// TIA Portal V15.1 export
// export: Created 2024-06-21T08:41:09.7541663Z, ExportSetting WithDefaults, DisplayName Totally Integrated Automation Portal, DisplayVersion V15.1 Update 5, DisplayName TIA Portal Openness, DisplayVersion V15.1 Update 5, DisplayName SINAMICS Startdrive Advanced, DisplayVersion V15.1, DisplayName G130, G150, S120, S150, SINAMICS MV, S210, DisplayVersion V15.1, DisplayName G110M, G120, G120C, G120D, G120P, DisplayVersion V15.1, DisplayName STEP 7 Professional, DisplayVersion V15.1 Update 5, DisplayName STEP 7 Safety, DisplayVersion V15.1, DisplayName WinCC Professional, DisplayVersion V15.1 Update 5, DisplayName SIMATIC Visualization Architect, DisplayVersion V15.1
FUNCTION "LGBLiftTable2Pos1S3Det-MoviFitFCPN-Config" : Void   // FC6651, FBD
TITLE = LMovUnit2Pos2Det2W2S-G120CU240PN-Config / LConfigMovUnit2Pos2W2S-G120PN / LGBLiftTable2Pos1S4Det-MoviFitFCPN-Config
{ S7_Optimized_Access := 'TRUE' }
AUTHOR : VCC
FAMILY : Control
NAME : Bit2Word
VERSION : 1.0
// =============================================================================
// Moves Configuration
// =============================================================================
// stored: AutoNumber false, IsIECCheckEnabled false, SetENOAutomatically False, UDAEnableTagReadback false
   VAR_INPUT
      C_ForceManual : Bool;   // Force Manual Enabled
      C_PosSetCheckUsed : Bool;   // 2nd Set Pos Check Used
      C_PosResCheckUsed : Bool;   // 2nd Set Pos Check Used
      C_AlarmResetUsed : Bool;   // Set position / If true, the Alarms will be stored untill reseted
      C_EnableMemBegin : Bool;   // Reset position / Enable memory Begin (Command Request is memorised until pos reached)
      C_EnIntlkAlm : Bool;   // Active / Enable interlock Alarm
      C_KeepPosition : Bool;   // Invisible / If true, the last position shall be kept ON and checked
      C_EnAlmDet : Bool;   // Object out of use / Enable Alarm
      C_EnableAlarmHW : Bool;   // Enable Alarm hardware (e.g. safetyswitch, motorprotector, detections)
      C_MotorProtectionNc : Bool;   // Motor Protection NC contact
      C_MotorProtectionUsed : Bool;   // Motor Protection used
      C_ReleaseBrakeUsed : Bool;   // Release brake used
      C_MotionStopUsed : Bool;   // Motion Stop used
      C_EnAlmOvertime : Bool;   // Interlock for Reset direction / Enable Overtime Alarm
      C_AlarmHighSeverity : Bool;   // Interlock alarm for Set direction / Alarm severity
      C_InitDirection : Bool;   // Initial direction
      C_HomePosIsUp : Bool;   // The home position of the lift table is up
      C_PosSetDelayTime : DInt;   // Set position delay timer / Set Position Delay Timer
      C_PosResDelayTime : DInt;   // Reset position delay timer / Reset Position Delay Timer
      C_DiscrTimeSetDet : DInt;   // Maximum Time (x1ms) between Set detections before creating alarm
      C_DiscrTimeResDet : DInt;   // Maximum Time (x1ms) between Res detections before creating alarm
      C_RunTimeMaxSetWarn : DInt;   // Maximum Time (x1ms) that the function may run (create overtime) / Maximum Time (x1ms) that the function may run (create Overtime)
      C_RunTimeMaxSetAlarm : DInt;   // Maximum Time (x1ms) that the function may run (create overtime) / Maximum Time (x1ms) that the function may run (create Overtime)
      C_RunTimeMaxResWarn : DInt;   // Maximum Time (x1ms) that the function may run (create overtime) / Maximum Time (x1ms) that the function may run (create Overtime)
      C_RunTimeMaxResAlarm : DInt;   // Maximum Time (x1ms) that the function may run (create overtime) / Maximum Time (x1ms) that the function may run (create Overtime)
      C_TimeAlmFilt : DInt;   // Timer before any actuator alarm will be active (welding..) / Timer before any actuator Alarm will be active (welding..)
      C_Ramp : Time;   // Ramp
      C_ReferenceMotorCurrent : Real;   // Reference value for current
      C_ReferenceDriveCurrent : Real;   // Reference value for drive
      C_HWSubInput : HW_SUBMODULE;   // I/O
      C_HWSubOutput : HW_SUBMODULE;   // I/O
      C_HWSubInputStatus : HW_SUBMODULE;   // I/O
   END_VAR
   VAR_IN_OUT
      IO_ConfigMoveUnit : "LiftTable2Pos1S3DetMoviFitFCPNConfig";   // Config
   END_VAR
BEGIN

REGION Network 1: **** 1 - Inputs **** Move Bit Config
   // Move Bit Config
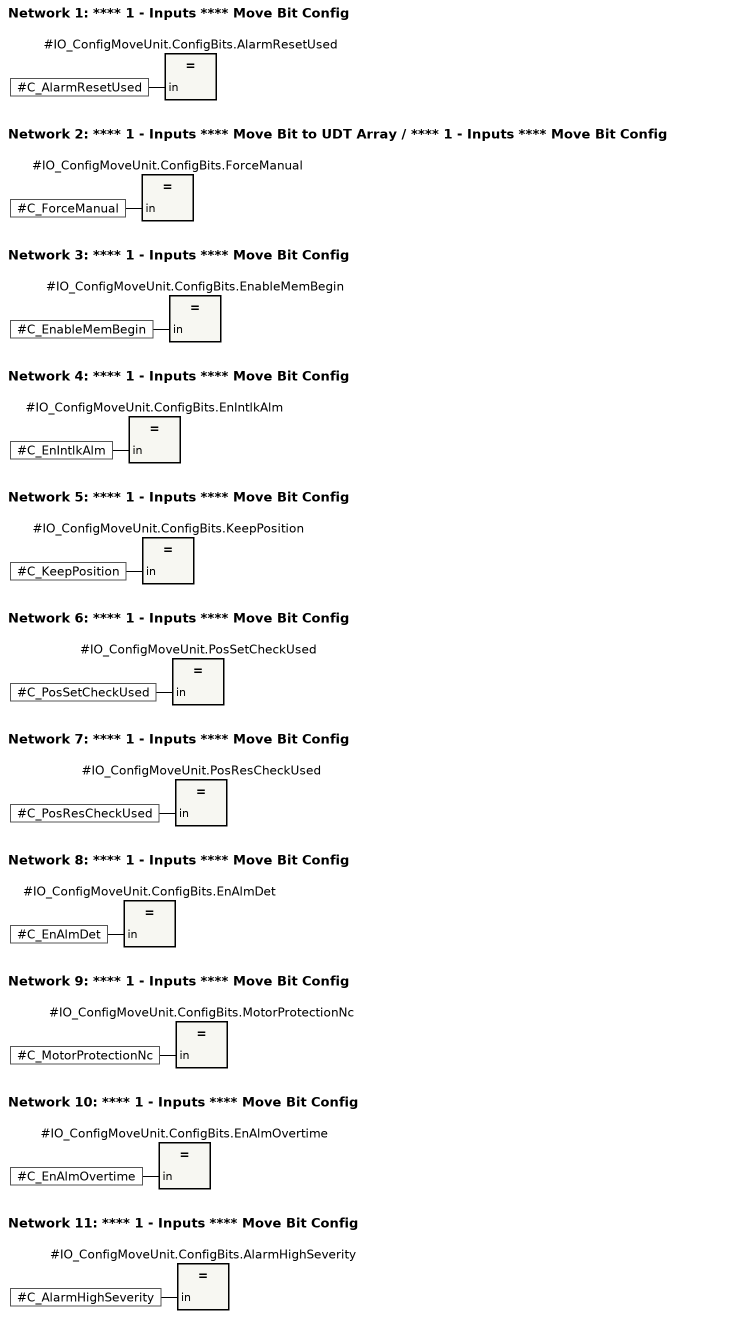
   #IO_ConfigMoveUnit.ConfigBits.AlarmResetUsed := #C_AlarmResetUsed;
END_REGION

REGION Network 2: **** 1 - Inputs **** Move Bit to UDT Array / **** 1 - Inputs **** Move Bit Config
   // Move Bit  to UDT Array
   #IO_ConfigMoveUnit.ConfigBits.ForceManual := #C_ForceManual;
END_REGION

REGION Network 3: **** 1 - Inputs **** Move Bit Config
   // Move Bit Config
   #IO_ConfigMoveUnit.ConfigBits.EnableMemBegin := #C_EnableMemBegin;
END_REGION

REGION Network 4: **** 1 - Inputs **** Move Bit Config
   // Move Bit Config
   #IO_ConfigMoveUnit.ConfigBits.EnIntlkAlm := #C_EnIntlkAlm;
END_REGION

REGION Network 5: **** 1 - Inputs **** Move Bit Config
   // Move Bit Config
   #IO_ConfigMoveUnit.ConfigBits.KeepPosition := #C_KeepPosition;
END_REGION

REGION Network 6: **** 1 - Inputs **** Move Bit Config
   // Move Bit Config
   #IO_ConfigMoveUnit.PosSetCheckUsed := #C_PosSetCheckUsed;
END_REGION

REGION Network 7: **** 1 - Inputs **** Move Bit Config
   // Move Bit Config
   #IO_ConfigMoveUnit.PosResCheckUsed := #C_PosResCheckUsed;
END_REGION

REGION Network 8: **** 1 - Inputs **** Move Bit Config
   // Move Bit Config
   #IO_ConfigMoveUnit.ConfigBits.EnAlmDet := #C_EnAlmDet;
END_REGION

REGION Network 9: **** 1 - Inputs **** Move Bit Config
   // Move Bit Config
   #IO_ConfigMoveUnit.ConfigBits.MotorProtectionNc := #C_MotorProtectionNc;
END_REGION

REGION Network 10: **** 1 - Inputs **** Move Bit Config
   // Move Bit Config
   #IO_ConfigMoveUnit.ConfigBits.EnAlmOvertime := #C_EnAlmOvertime;
END_REGION

REGION Network 11: **** 1 - Inputs **** Move Bit Config
   // Move Bit Config
   #IO_ConfigMoveUnit.ConfigBits.AlarmHighSeverity := #C_AlarmHighSeverity;
END_REGION

REGION Network 12: **** 1 - Inputs **** Move Bit Config
   // Move Bit Config
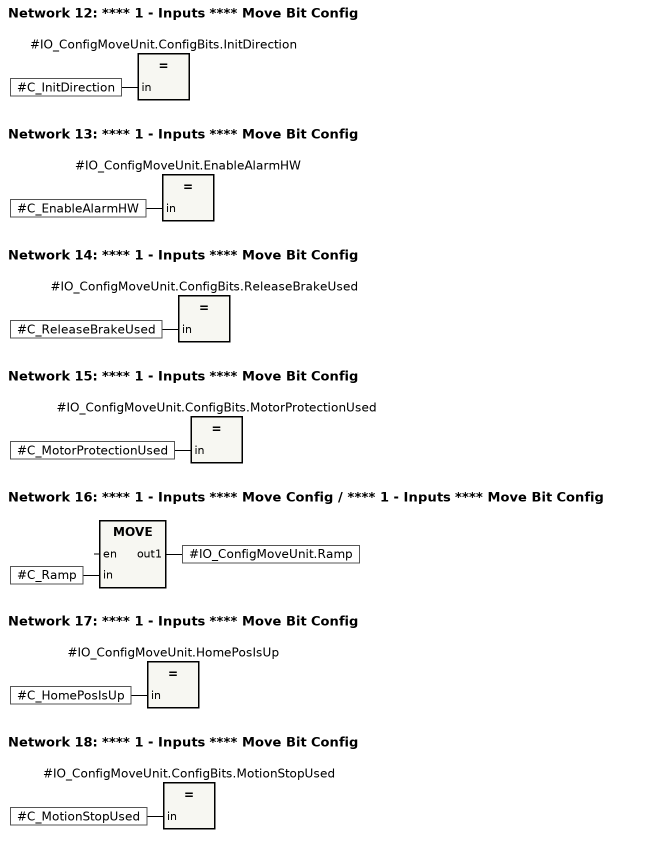
   #IO_ConfigMoveUnit.ConfigBits.InitDirection := #C_InitDirection;
END_REGION

REGION Network 13: **** 1 - Inputs **** Move Bit Config
   // Move Bit Config
   #IO_ConfigMoveUnit.EnableAlarmHW := #C_EnableAlarmHW;
END_REGION

REGION Network 14: **** 1 - Inputs **** Move Bit Config
   // Move Bit Config
   #IO_ConfigMoveUnit.ConfigBits.ReleaseBrakeUsed := #C_ReleaseBrakeUsed;
END_REGION

REGION Network 15: **** 1 - Inputs **** Move Bit Config
   // Move Bit Config
   #IO_ConfigMoveUnit.ConfigBits.MotorProtectionUsed := #C_MotorProtectionUsed;
END_REGION

REGION Network 16: **** 1 - Inputs **** Move Config / **** 1 - Inputs **** Move Bit Config
   // Move Config
   #IO_ConfigMoveUnit.Ramp := #C_Ramp;
END_REGION

REGION Network 17: **** 1 - Inputs **** Move Bit Config
   // Move Bit Config
   #IO_ConfigMoveUnit.HomePosIsUp := #C_HomePosIsUp;
END_REGION

REGION Network 18: **** 1 - Inputs **** Move Bit Config
   // Move Bit Config
   #IO_ConfigMoveUnit.ConfigBits.MotionStopUsed := #C_MotionStopUsed;
END_REGION

NETWORK
TITLE = **** 1 Inputs **** Move Config UDT
// Move Config
      L     #C_PosSetDelayTime;
      T     #IO_ConfigMoveUnit.PosSetDelayTime;
      L     #C_PosResDelayTime;
      T     #IO_ConfigMoveUnit.PosResDelayTime;
      L     #C_RunTimeMaxSetWarn;
      T     #IO_ConfigMoveUnit.RunTimeMaxSetWarn;
      L     #C_RunTimeMaxSetAlarm;
      T     #IO_ConfigMoveUnit.RunTimeMaxSetAlm;
      L     #C_RunTimeMaxResWarn;
      T     #IO_ConfigMoveUnit.RunTimeMaxResWarn;
      L     #C_RunTimeMaxResAlarm;
      T     #IO_ConfigMoveUnit.RunTimeMaxResAlm;
      L     #C_TimeAlmFilt;
      T     #IO_ConfigMoveUnit.TimeAlmFilt;
      L     #C_ReferenceMotorCurrent;
      T     #IO_ConfigMoveUnit.ReferenceMotorCurrent;
      L     #C_ReferenceDriveCurrent;
      T     #IO_ConfigMoveUnit.ReferenceDriveCurrent;
      L     #C_HWSubInput;
      T     #IO_ConfigMoveUnit.HWSubInput;
      L     #C_HWSubOutput;
      T     #IO_ConfigMoveUnit.HWSubOutput;
      L     #C_HWSubInputStatus;
      T     #IO_ConfigMoveUnit.HWSubInputStatus;




NETWORK
TITLE = **** 1 Inputs **** Move Config UDT
// Move Config
      A     "TRUE";
      L     #C_DiscrTimeSetDet;
      T     #IO_ConfigMoveUnit.DiscrTimeSetDet;
      L     #C_DiscrTimeResDet;
      T     #IO_ConfigMoveUnit.DiscrTimeResDet;

      L     0.0;
      T     #IO_ConfigMoveUnit.ReferenceMotorRPM;
      L     0.0;
      T     #IO_ConfigMoveUnit.RatioGearbox;
      L     0.0;
      T     #IO_ConfigMoveUnit.Diameter;
      L     0.0;
      T     #IO_ConfigMoveUnit.Acceleration;
END_FUNCTION
